Fanuc KAREL source: compact_preamble.KL

PROGRAM KA00134
%NOLOCKGROUP
VAR
SRC : ARRAY[2] OF SHORT
DST:REAL
BEGIN
SRC[1]=2
DST=(SRC[1])
END KA00134
